TYPE ST_PackML_ControlX :
    STRUCT
        CurrentMode  : E_PMLUnitMode;
        ModeCommand  : E_PMLUnitMode;
        CurrentState : E_PMLState;
        StateCommand : E_PMLCommand;
        ModeNames    : ARRAY[0..31] OF STRING;
    END_STRUCT
END_TYPE

(* stored: Version 1.1.0.1
   DUT ST_PackML_ControlX: Id {a3390312-c7bc-4c83-b9cf-ef4e77bd2c27} *)
